(*

short summary
=================
This class implements the interface :ref:`I64BitTimeAssertions`. 
It provides the assert statements for the data type ``LTIME``

.. <legal notes>

legal notes
=================
| SPDX-FileCopyrightText: © 2022 ekvip automation GmbH <info@ekvip.de>
| SPDX-License-Identifier: Apache-2.0
| For details check: Apache-2.0_

.. _Apache-2.0: https://www.apache.org/licenses/LICENSE-2.0

.. </legal notes>

methods and properties
=========================

*)

{attribute 'reflection'}
FUNCTION_BLOCK INTERNAL LongTimeAssertions EXTENDS AbstactAssertion IMPLEMENTS I64BitTimeAssertions
VAR CONSTANT
	(* maximum value for the data type ``LTIME`` *)
	MAX_TIME	:LTIME := TO_LTIME(16#FFFF_FFFF_FFFF_FFFF);
END_VAR

(*

short summary
=================
This abstract property returns the class name of the concrete object, 
It's for debugging purpose

.. <legal notes>

legal notes
=================
| SPDX-FileCopyrightText: © 2022 ekvip automation GmbH <info@ekvip.de>
| SPDX-License-Identifier: Apache-2.0
| For details check: Apache-2.0_

.. _Apache-2.0: https://www.apache.org/licenses/LICENSE-2.0

.. </legal notes>

*)

PROPERTY className :ClassName
GET
className := 'CNM_AssertionInterfaceLib.LongTimeAssertions';
END_GET
END_PROPERTY

(*

short summary
=================
This method returns the passed time since the timestamp was created

.. <legal notes>

legal notes
=================
| SPDX-FileCopyrightText: © 2022 ekvip automation GmbH <info@ekvip.de>
| SPDX-License-Identifier: Apache-2.0
| For details check: Apache-2.0_

.. _Apache-2.0: https://www.apache.org/licenses/LICENSE-2.0

.. </legal notes>

parameters
=================
:return: passed time since ``startTime``

*)

METHOD PROTECTED getTimePassed :LTIME
VAR_INPUT
	(* timestamp start *)
	startTime	:LTIME;
END_VAR
VAR
	(* current time to calculate the passed time *)
	currentTime	:LTIME;
END_VAR
currentTime := LTIME();
IF (currentTime > startTime) THEN
	getTimePassed := (currentTime - startTime);
ELSE
	getTimePassed := ((THIS^.MAX_TIME - startTime) + currentTime);
END_IF
END_METHOD

(*

short summary
=================
This assertion method checks whether time has elapsed since the timestamp time

.. <legal notes>

legal notes
=================
| SPDX-FileCopyrightText: © 2022 ekvip automation GmbH <info@ekvip.de>
| SPDX-License-Identifier: Apache-2.0
| For details check: Apache-2.0_

.. _Apache-2.0: https://www.apache.org/licenses/LICENSE-2.0

.. </legal notes>

parameters
=================

*)

METHOD timeHasExpired
VAR_INPUT
	(* start time you get it with ``LTIME()`` *)
	timestamp		:LTIME;
	(* timeout like ``lt#300ms`` *)
	expiringTime	:LTIME;
	(* message if the assertion is false *)
	message			:AssertMessage;
END_VAR
VAR
	(* measured passed time *)
	passedTime		:LTIME;
END_VAR
passedTime := THIS^.getTimePassed(timestamp);
IF (passedTime < expiringTime) THEN
	THIS^.assertionWasWrong(
		message			:= message,
		additionalText	:= THIS^.getDebugInfo('timeHasExpired')
	);	
END_IF
END_METHOD

(*

short summary
=================
This assertion method checks that the time since the timestamp time has not yet elapsed

.. <legal notes>

legal notes
=================
| SPDX-FileCopyrightText: © 2022 ekvip automation GmbH <info@ekvip.de>
| SPDX-License-Identifier: Apache-2.0
| For details check: Apache-2.0_

.. _Apache-2.0: https://www.apache.org/licenses/LICENSE-2.0

.. </legal notes>

parameters
=================

*)

METHOD timeHasNotExpired
VAR_INPUT
	(* start time you get it with ``LTIME()`` *)
	timestamp		:LTIME;
	(* timeout like ``lt#300ms`` *)
	expiringTime	:LTIME;
	(* message if the assertion is false *)
	message			:AssertMessage;
END_VAR
VAR
	(* measured passed time *)
	passedTime		:LTIME;
END_VAR
passedTime := THIS^.getTimePassed(timestamp);
IF (passedTime >= expiringTime) THEN
	THIS^.assertionWasWrong(
		message			:= message,
		additionalText	:= THIS^.getDebugInfo('timeHasNotExpired')
	);	
END_IF
END_METHOD

(*

short summary
=================
This assertion method checks if the current value is equal to the expected value

.. <legal notes>

legal notes
=================
| SPDX-FileCopyrightText: © 2022 ekvip automation GmbH <info@ekvip.de>
| SPDX-License-Identifier: Apache-2.0
| For details check: Apache-2.0_

.. _Apache-2.0: https://www.apache.org/licenses/LICENSE-2.0

.. </legal notes>

parameters
=================

*)

METHOD valueIsEqualTo
VAR_INPUT
	(* current value to check *)
	currentValue	:LTIME;
	(* expected value to compare *)
	expectedValue	:LTIME;
	(* message if the assertion is false *)
	message	:AssertMessage;
END_VAR
IF (currentValue <> expectedValue) THEN
	THIS^.assertionWasWrong(
		message			:= message,
		additionalText	:= THIS^.getDebugInfo('valueIsEqualTo')
	);	
END_IF
END_METHOD

(*

short summary
=================
This assertion method checks if the current value is greater than the less value

.. <legal notes>

legal notes
=================
| SPDX-FileCopyrightText: © 2022 ekvip automation GmbH <info@ekvip.de>
| SPDX-License-Identifier: Apache-2.0
| For details check: Apache-2.0_

.. _Apache-2.0: https://www.apache.org/licenses/LICENSE-2.0

.. </legal notes>

parameters
=================

*)

METHOD valueIsGreaterThan
VAR_INPUT
	(* current value to check *)
	currentValue	:LTIME;
	(* less than lower limit *)
	lessValue		:LTIME;
	(* message if the assertion is false *)
	message	: AssertMessage;
END_VAR
IF (currentValue <= lessValue) THEN
	THIS^.assertionWasWrong(
		message			:= message,
		additionalText	:= THIS^.getDebugInfo('valueIsGreaterThan')
	);	
END_IF
END_METHOD

(*

short summary
=================
This assertion method checks if the current value is inside a limit

.. attention:: 
	limits are included: ``valueIsInRangeOf(t#3ms,t#3ms ,t#3ms)`` is a true assertion

.. <legal notes>

legal notes
=================
| SPDX-FileCopyrightText: © 2022 ekvip automation GmbH <info@ekvip.de>
| SPDX-License-Identifier: Apache-2.0
| For details check: Apache-2.0_

.. _Apache-2.0: https://www.apache.org/licenses/LICENSE-2.0

.. </legal notes>

parameters
=================

*)

METHOD valueIsInRangeOf
VAR_INPUT
	(* lower limit for the current value *)
	lowerLimit		:LTIME;
	(* current value to check *)
	currentValue	:LTIME;
	(* upper limit for the current value *)
	upperLimit		:LTIME;
	(* message if the assertion is false *)
	message			:AssertMessage;
END_VAR
VAR
	(* additional information for the callback function *)
	additionalText	:Tc2_System.T_MaxString;
END_VAR
IF ((currentValue < lowerLimit) OR (currentValue > upperLimit)) THEN
	THIS^.assertionWasWrong(
		message			:= message,
		additionalText	:= THIS^.getDebugInfo('valueIsInRangeOf')
	);	
END_IF
END_METHOD

(*

short summary
=================
This assertion method checks if the current value is less than the greater value

.. <legal notes>

legal notes
=================
| SPDX-FileCopyrightText: © 2022 ekvip automation GmbH <info@ekvip.de>
| SPDX-License-Identifier: Apache-2.0
| For details check: Apache-2.0_

.. _Apache-2.0: https://www.apache.org/licenses/LICENSE-2.0

.. </legal notes>

parameters
=================

*)

METHOD valueIsLessThan
VAR_INPUT
	(* current value to check *)
	currentValue	:LTIME;
	(* greater than upper limit *)
	greaterValue	:LTIME;
	(* message if the assertion is false *)
	message			:AssertMessage;
END_VAR
IF (currentValue >= greaterValue) THEN
	THIS^.assertionWasWrong(
		message			:= message,
		additionalText	:= THIS^.getDebugInfo('valueIsLessThan')
	);	
END_IF
END_METHOD

(*

short summary
=================
This assertion method checks if the current value is less than or equal to the maximum value

.. <legal notes>

legal notes
=================
| SPDX-FileCopyrightText: © 2022 ekvip automation GmbH <info@ekvip.de>
| SPDX-License-Identifier: Apache-2.0
| For details check: Apache-2.0_

.. _Apache-2.0: https://www.apache.org/licenses/LICENSE-2.0

.. </legal notes>

parameters
=================

*)

METHOD valueIsMax
VAR_INPUT
	(* current value to check *)
	currentValue	:LTIME;
	(* upper limit for the current value *)
	maximumValue	:LTIME;
	(* message if the assertion is false *)
	message			:AssertMessage;
END_VAR
IF (currentValue > maximumValue) THEN
	THIS^.assertionWasWrong(
		message			:= message,
		additionalText	:= THIS^.getDebugInfo('valueIsMax')
	);	
END_IF
END_METHOD

(*

short summary
=================
This assertion method checks if the current value is greater than or equal to the minimum value

.. <legal notes>

legal notes
=================
| SPDX-FileCopyrightText: © 2022 ekvip automation GmbH <info@ekvip.de>
| SPDX-License-Identifier: Apache-2.0
| For details check: Apache-2.0_

.. _Apache-2.0: https://www.apache.org/licenses/LICENSE-2.0

.. </legal notes>

parameters
=================

*)

METHOD valueIsMin
VAR_INPUT
	(* current value to check *)
	currentValue	:LTIME;
	(* lower limit for the current value *)
	minimumValue	:LTIME;
	(* message if the assertion is false *)
	message			:AssertMessage;
END_VAR
IF (currentValue < minimumValue) THEN
	THIS^.assertionWasWrong(
		message			:= message,
		additionalText	:= THIS^.getDebugInfo('valueIsMin')
	);	
END_IF
END_METHOD

(*

short summary
=================
This assertion method checks if the current value is not equal to the unexpected value

.. <legal notes>

legal notes
=================
| SPDX-FileCopyrightText: © 2022 ekvip automation GmbH <info@ekvip.de>
| SPDX-License-Identifier: Apache-2.0
| For details check: Apache-2.0_

.. _Apache-2.0: https://www.apache.org/licenses/LICENSE-2.0

.. </legal notes>

parameters
=================

*)

METHOD valueIsNotEqualTo
VAR_INPUT
	(* current value to check *)
	currentValue	:LTIME;
	(* unexpected value to compare *)
	unexpectedValue	:LTIME;
	(* message if the assertion is false *)
	message			:AssertMessage;
END_VAR
IF (currentValue = unexpectedValue) THEN
	THIS^.assertionWasWrong(
		message			:= message,
		additionalText	:= THIS^.getDebugInfo('valueIsNotEqualTo')
	);	
END_IF
END_METHOD

END_FUNCTION_BLOCK

(* stored: Version 1.1.0.1, ProductVersion 3.1.4024.11
   POU LongTimeAssertions: Id {b2dffb11-d7c3-4f48-a098-511f1dfa695f}, SpecialFunc None
   Property className: Id {a7a60e8e-a881-4459-87f8-4d07907353b2}
   Get Get: Id {2d5466ae-3b32-4ca1-8840-e510a2134017}
   Method getTimePassed: Id {98cacde6-c133-41f0-a513-7f1463cae644}
   Method timeHasExpired: Id {6891eb87-d5b4-488e-bf83-9d469864b96e}
   Method timeHasNotExpired: Id {da85888b-78c7-4d71-80e8-8a55ba4d9390}
   Method valueIsEqualTo: Id {50e44fd4-63ac-4bb7-a07e-ae12f49aed51}
   Method valueIsGreaterThan: Id {aa0a2c06-f32c-419f-8ebe-46fa6928017c}
   Method valueIsInRangeOf: Id {6bbce859-0dae-4859-8d9f-68a3dbabe567}
   Method valueIsLessThan: Id {13e6d15c-a90d-43e0-8be0-e06fb427ab23}
   Method valueIsMax: Id {e1954234-e88d-495e-aebb-adf539b494bb}
   Method valueIsMin: Id {e234b0d6-fff0-447a-9b24-0cfdbca2add1}
   Method valueIsNotEqualTo: Id {75c749a8-5a23-45bd-b6b5-80fbd9ad34fc} *)
